// TIA Portal V18 export
TYPE "DT_FML_PRM_FILE"
// stored: IsFailsafeCompliant false
   STRUCT
      Control : Int;
      BitSequenceNr : Int;
      Data : Array[1..6] of Byte;
   END_STRUCT;
END_TYPE
